{attribute 'qualified_only'}
VAR_GLOBAL
	cMaxNumberOfEvent:UINT; //
	
	
	
END_VAR

(* stored: Version 1.1.0.1, ProductVersion 3.1.4024.11
   GVL GVL_EventLogger: Id {5524e0ab-d51e-4a76-bd9b-c2deb3e8a064} *)
